FUNCTION Pow2 : LREAL
VAR_INPUT
	number : LREAL;
END_VAR

Pow2 := number * number;

END_FUNCTION

(* stored: Version 1.1.0.1
   POU Pow2: Id {37161c21-4d66-02e2-2232-88e65cb4eecd}, SpecialFunc None *)
